Fanuc KAREL source: kt00104.KL

-- PROVISIONAL review KL for V940-1; original PC SHA256 a70d482a00bda3576fb96a5110b89420d79c437bc076844c21b889d29b3d1d98
-- Incomplete behavior may be omitted. Consult companion uncertainty JSON. Do not deploy.
PROGRAM KT00104
%NOLOCKGROUP
VAR
  I1 : INTEGER
  OUT : REAL
-- UNRESOLVED_DECL H2 type=002017
BEGIN
  -- V9_ZERO_TABLE_METADATA_HINT layout=0001; no indexed target words; source/name/runtime held
  -- UNRESOLVED_PC offsets 5-16; opcodes 2E,23
  -- UNRESOLVED_PC offsets 21-35; opcodes 2E,22,9D,33,B4
  -- UNRESOLVED_PC offsets 40-66; opcodes 21,22,9D,33,B3,64,29,64,29,6C,23
  -- UNRESOLVED_PC offsets 71-75; opcodes 7F
END KT00104
